FUNCTION_BLOCK ValveDynamics
VAR_INPUT
	udcv_IN : LREAL;
	wn : LREAL := 30.0;
	dr : LREAL := 0.7;
END_VAR
VAR_OUTPUT
	DynamicValve : LREAL;
END_VAR
VAR
	fDeltaTime : LREAL := 0.001;
	fAcceleration : LREAL;
	fbVelocity : TimeIntegrator := (fInit := 0.0);
	fbPosition : TimeIntegrator := (fInit := 0.0);
	a : LREAL;
	b : LREAL;
END_VAR
VAR CONSTANT
END_VAR

//Timer := Timer + 0.001;

////Valve opening signal is sent through this
//DynamicValve := cst1*EXP(-21*Timer)*SIN(cst2*Timer);

IF (wn = 0.0) THEN
	RETURN;
END_IF

a := 1/EXPT(wn, 2.0);
b := dr/wn;

fAcceleration := (udcv_IN - 2*fbVelocity.fOut*b - fbPosition.fOut)/a;

fbVelocity(
	fIn := fAcceleration,
	fStepTime := fDeltaTime,
);

fbPosition(
	fIn := fbVelocity.fOut,
	fStepTime := fDeltaTime,
	bEnableLimits := TRUE,
	fMinVal := -1.0,
	fMaxVal := 1.0,
	fOut => DynamicValve
);

END_FUNCTION_BLOCK

(* stored: Version 1.1.0.1, ProductVersion 3.1.4024.9
   POU ValveDynamics: Id {bdd402cd-9955-422d-9429-c814b00ee090}, SpecialFunc None *)
